FUNCTION_BLOCK PrintStatus
  (* Standard: 61499-2 *)
  (* Version 0.1, 2017-00-16, hpea485, UOA *)
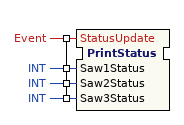
  EVENT_INPUT
    StatusUpdate WITH Saw1Status, Saw2Status, Saw3Status;
  END_EVENT
  VAR_INPUT
    Saw1Status : INT;
    Saw2Status : INT;
    Saw3Status : INT;
  END_VAR
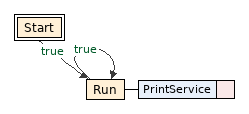
  EC_STATES
    Start;
    Run : PrintService;
  END_STATES
  EC_TRANSITIONS
    Start TO Run := true;
    Run TO Run := true;
  END_TRANSITIONS
  ALGORITHM PrintService IN C:
// OFF 0
// RUNNING 1
// WEIGHT -1
// LASER -2
// STALL -3
// SPEED -4

if(me->inputEvents.event.StatusUpdate) {
	printf("Saw 1: ");
	switch(me->Saw1Status) {
		case 0:
			printf("OFF          ");
			break;
		case 1:
			printf("RUNNING      ");
			break;
		case -1:
			printf("ERR:SAWDUST  ");
			break;
		case -2:
			printf("ERR:PROXIMITY");
			break;
		case -3:
			printf("ERR:STALL    ");
			break;
		case -4:
			printf("ERR:JITTER   ");
			break;
		default:
			printf("ERR:UNKNOWN  ");
	}
	printf("\t");

	printf("Saw 2: ");
	switch(me->Saw2Status) {
		case 0:
			printf("OFF          ");
			break;
		case 1:
			printf("RUNNING      ");
			break;
		case -1:
			printf("ERR:SAWDUST  ");
			break;
		case -2:
			printf("ERR:PROXIMITY");
			break;
		case -3:
			printf("ERR:STALL    ");
			break;
		case -4:
			printf("ERR:JITTER   ");
			break;
		default:
			printf("ERR:UNKNOWN  ");
	}
	printf("\t");

	printf("Saw 3: ");
	switch(me->Saw3Status) {
		case 0:
			printf("OFF          ");
			break;
		case 1:
			printf("RUNNING      ");
			break;
		case -1:
			printf("ERR:SAWDUST  ");
			break;
		case -2:
			printf("ERR:PROXIMITY");
			break;
		case -3:
			printf("ERR:STALL    ");
			break;
		case -4:
			printf("ERR:JITTER   ");
			break;
		default:
			printf("ERR:UNKNOWN  ");
	}
	printf("\n");

}
  END_ALGORITHM
END_FUNCTION_BLOCK
